(* CODESYS project ex_02.project

Project tree, tasks and I/O mapping:
  Device : CODESYS Control Win V3, 3S - Smart Software Solutions GmbH, version 3.5.20.50
    application Application
      libraries: Standard, 3.5.18.0 (System)
      task MainTask (cyclic, interval t#20ms, priority 1) calls PLC_PRG
      program PLC_PRG [ST]
*)

// Device/Application/PLC_PRG
PROGRAM PLC_PRG
VAR
	button1:BOOL;
	button2:BOOL;
	motor:BOOL;
END_VAR

IF (button1=FALSE AND button2=TRUE) OR (button1=TRUE AND button2=FALSE) THEN
	motor:=TRUE;
ELSE
	motor:=FALSE;
END_IF

END_PROGRAM
